//{{V2}}
DATA_BLOCK DB10

AUTHOR:nb
FAMILY:nb
NAME:nb
VERSION:1.0


FB1

BEGIN

       SP:=0.000000e+00
       PV:=0.000000e+00
       K_P:=0.000000e+00
       K_I:=FALSE
       CTRL:=0.000000e+00
       E:=0.000000e+00
END_DATA_BLOCK
